PROGRAM Rotation
VAR
//Outputs: Power for Limit switches, Home Sensors, etc.
    //bPowerSwitchesAxis1 AT %Q*: BOOL:= TRUE;
    bFwdLimitPower AT %Q* : BOOL := TRUE;
    bBwdLimitPower AT %Q* : BOOL := TRUE;
    bEnable : BOOL := TRUE;
//Hardware interlocks
    //bInterlockFwdOK AT %I*: BOOL;
END_VAR

//Initial parameters of an Axis
(*IF _TaskInfo[fbGetCurTaskIndex.index].FirstCycle THEN
    //Initial default values:
    GVL.astAxes[1].stConfig.eHomeSeq := 0;
    GVL.astAxes[1].stConfig.fHomePosition := 0.0;
    GVL.astAxes[1].stConfig.fHomeFinishDistance := 0.0;
    GVL.astAxes[1].stConfig.eRestorePosition := E_RestorePosition.eRestoreWithoutHome;
END_IF*)
astAxes[AXIS_ROTATION].stControl.bEnable := bEnable;
astAxes[AXIS_ROTATION].stInputs.bLimitBwd := TRUE;
astAxes[AXIS_ROTATION].stInputs.bLimitFwd := TRUE;
//Define ACTIONS() or write exclusive code for an specific axis.
(*Eg. Stop when temperature reaches certain values, reduce speed if  a signal is activated, etc.
Eg. GVL.astAxes[x].stControl.bInterlockFwd := NOT bInterlockFwdOK;*)

END_PROGRAM

(* stored: Version 1.1.0.1, ProductVersion 3.1.4024.12
   POU Rotation: Id {83b74736-0e2a-4820-b07c-7378d567dc02}, SpecialFunc None *)
